(* CoDeSys 2.3 export: GETEEP_P3.EXP *)

(* POU 05_Basic_Calc/eeprom_operations/getEEP_P3, ST *)
FUNCTION getEEP_P3 : INT
VAR_INPUT
	EEP_num				: INT;
END_VAR
VAR
	EEP_PAGE3_OFFSET	: INT		:= 768;
END_VAR
getEEP_P3	:= EEP_num - EEP_PAGE3_OFFSET;
END_FUNCTION
